TYPE ST_MoverData :
STRUCT
	id : UDINT;
	pos : LREAL;
	status : INT;
	assigned : BOOL;
END_STRUCT
END_TYPE

(* stored: Version 1.1.0.1, ProductVersion 3.1.4026.12
   DUT ST_MoverData: Id {c098c46e-b095-433c-ad89-ba10fd5ca898} *)
